TYPE CmpWMxFQAGate :
STRUCT
	Framework: Framework;
	StatusInCycleAuto: BOOL;
	FreeRunCycleStop: BOOL;
	Config: CmpWmxFQAGateConfig;
END_STRUCT
END_TYPE

(* stored: Version 1.1.0.1, ProductVersion 3.1.4024.6
   DUT CmpWMxFQAGate: Id {80e2ffa2-c332-42ac-8ae7-663df829c724} *)
